INTERFACE I_DeserializerObjectForwardEnumerator EXTENDS I_Disposable

PROPERTY PUBLIC Current : I_Deserializer
GET
END_GET
END_PROPERTY

PROPERTY IsValid : BOOL
GET
END_GET
END_PROPERTY

PROPERTY Key : T_MAXSTRING
GET
END_GET
END_PROPERTY

METHOD MoveNext : BOOL
VAR_INPUT
END_VAR
END_METHOD

END_INTERFACE

(* stored: Version 1.1.0.1, ProductVersion 3.1.4024.12
   Itf I_DeserializerObjectForwardEnumerator: Id {e7c955a7-2970-0b7e-166a-b0da059af6ce}
   Property Current: Id {653422f8-c101-0e77-0e09-8e5e6e9f092b}
   Get Get: Id {711fe33b-09fe-0eab-33ca-529e23f3dafa}
   Property IsValid: Id {4ddd6a3b-518d-08bb-2e51-bc08f09ac266}
   Get Get: Id {b7b2f816-5331-0bbe-2210-1c0b76a1a7cb}
   Property Key: Id {bb052cff-9bd5-02ab-149e-61ee39b2aef3}
   Get Get: Id {5d023078-ac51-00b5-3a45-d0d2ef14e7b8}
   Method MoveNext: Id {e81ada67-cbb4-04ce-0f2e-f070b7cade7a} *)
